FUNCTION_BLOCK FB_HE_SATT_FilterSelection
VAR
    iFilterHolder1 : I_HE_SATT_FilterHolder;
    iFilterHolder2 : I_HE_SATT_FilterHolder;
    iFilterHolder3 : I_HE_SATT_FilterHolder;
    iFilterHolder4 : I_HE_SATT_FilterHolder;
    iFilterHolder5 : I_HE_SATT_FilterHolder;
//     iCalculateSiliconThickness : I_CalculateThickness;
//     iCalculateDiamondThickness : I_CalculateThickness;
//     iCalculateGermaniumThickness : I_CalculateThickness;
END_VAR


METHOD FB_Init: BOOL
VAR_INPUT
    bInitRetains: BOOL; // TRUE: the retain variables are initialized (reset warm / reset cold)
    bInCopyCode: BOOL;  // TRUE: the instance will be copied to the copy code afterward (online change)
    iFilterHolder1 : I_HE_SATT_FilterHolder;
    iFilterHolder2 : I_HE_SATT_FilterHolder;
    iFilterHolder3 : I_HE_SATT_FilterHolder;
    iFilterHolder4 : I_HE_SATT_FilterHolder;
    iFilterHolder5 : I_HE_SATT_FilterHolder;
//     iCalculateSiliconThickness : I_CalculateThickness;
//     iCalculateDiamondThickness : I_CalculateThickness;
//     iCalculateGermaniumThickness : I_CalculateThickness;
END_VAR

THIS^.iFilterHolder1 := iFilterHolder1;
THIS^.iFilterHolder2 := iFilterHolder2;
THIS^.iFilterHolder3 := iFilterHolder3;
THIS^.iFilterHolder4 := iFilterHolder4;
THIS^.iFilterHolder5 := iFilterHolder5;
// THIS^.iCalculateSiliconThickness := iCalculateSiliconThickness;
// THIS^.iCalculateDiamondThickness := iCalculateDiamondThickness;
// THIS^.iCalculateGermaniumThickness := iCalculateGermaniumThickness;
END_METHOD


METHOD PUBLIC GetFilterPositions
VAR_INPUT
    fRequestedTransmission : LREAL; // [1]
    fPhotonEnergy : LREAL; // [eV]
    eRoundingMode : E_HE_SATT_RoundingMode;
END_VAR
VAR_OUTPUT
    fPosition1 : LREAL; // [mm]
    fPosition2 : LREAL; // [mm]
    fPosition3 : LREAL; // [mm]
    fPosition4 : LREAL; // [mm]
    fPosition5 : LREAL; // [mm]
    bError : BOOL;
    sError : T_MaxString;
END_VAR
VAR
    fSiliconThicknessRequired : LREAL;
    fDiamondThicknessRequired : LREAL;
END_VAR

// THIS^.iCalculateSiliconThickness.Calculate(
//     fDesiredTransmission := fRequestedTransmission,
//     fPhotonEnergy := fPhotonEnergy,
//     fThickness => fSiliconThicknessRequired
// );

IF fSiliconThicknessRequired < 200 THEN
//     THIS^.iCalculateDiamondThickness.Calculate(
//         fDesiredTransmission := fRequestedTransmission,
//         fPhotonEnergy := fPhotonEnergy,
//         fThickness => fDiamondThicknessRequired
//     );
    // Lookup which diamond filter is the closest one to the calcuated thickness accounting for the rounding mode.
    // Then give the positions (1-5) than would put the closest thickness diamond filters in the path of the beam.
    fPosition3 := 0.0; // 0.0 is defined as the OUT position.
    fPosition4 := 0.0; // 0.0 is defined as the OUT position.
    fPosition5 := 0.0; // 0.0 is defined as the OUT position.



ELSIF fSiliconThicknessRequired >= 200 AND fSiliconThicknessRequired < 6000 THEN
    // some procedure
ELSE
    // some procedure
END_IF
END_METHOD

END_FUNCTION_BLOCK

(* stored: Version 1.1.0.1
   POU FB_HE_SATT_FilterSelection: Id {03a9882a-fdb5-4066-a35a-05d3adec64d5}, SpecialFunc None
   Method FB_Init: Id {ddca28cb-2ee8-4e73-9fb8-aaad32671d0b}
   Method GetFilterPositions: Id {44eb97cc-a97a-4da8-9e85-294a95813109} *)
